TYPE ST_Monitoring :
STRUCT
	astMonitoringGlobal		: ARRAY[0..CONST.iMaxIdxMonitoring] OF ST_Data_Item;				// general/global monitoring
	astMonitoringModule		: ARRAY[0..E_Module.eModule_nMaxIdx] OF ST_Monitoring_Module;		// module monitoring
	astMonitoringStation	: ARRAY[0..E_Station.eStation_nMaxIdx] OF ST_Monitoring_Station;	// station monitoring
END_STRUCT
END_TYPE

(* stored: Version 1.1.0.1, ProductVersion 3.1.4024.12
   DUT ST_Monitoring: Id {23eb01c2-013a-42a1-9379-2c4028157f83} *)
